Fanuc KAREL source: CNC_DYN_DISP.kl

PROGRAM T
%NOLOCKGROUP
VAR
 v0 : INTEGER
 v1 : INTEGER
 v2 : STRING[40]
 v3 : INTEGER
BEGIN
 CNC_DYN_DISP(v0, v1, v2, v3)
END T
